{attribute 'TcGenerated'}
{attribute 'no-analysis'}
{attribute 'linkalways'}
// This function has been automatically generated from the project information.
VAR_GLOBAL CONSTANT
	{attribute 'const_non_replaced'}
	stLibVersion_Logging_file_library : ST_LibVersion := (iMajor := 0, iMinor := 0, iBuild := 1, iRevision := 1, nFlags := 0, sVersion := '0.0.1.1');
END_VAR

(* stored: Version 1.1.0.1, ProductVersion 3.1.4024.13
   GVL Global_Version: Id {62f2c78a-f3d5-0acd-0a64-61dfe36ef816} *)
